PROGRAM P5_00_MAIN
VAR

END_VAR

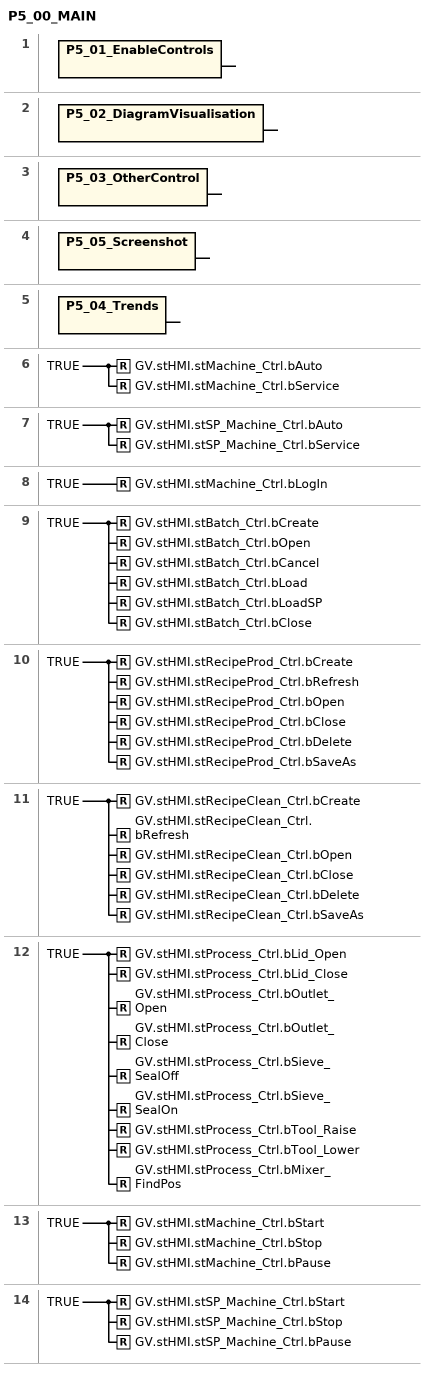
// NETWORK 1
P5_01_EnableControls();

// NETWORK 2
P5_02_DiagramVisualisation();

// NETWORK 3
P5_03_OtherControl();

// NETWORK 4
P5_05_Screenshot();

// NETWORK 5
P5_04_Trends();

// NETWORK 6
GV.stHMI.stMachine_Ctrl.bAuto R= TRUE;
GV.stHMI.stMachine_Ctrl.bService R= TRUE;

// NETWORK 7
GV.stHMI.stSP_Machine_Ctrl.bAuto R= TRUE;
GV.stHMI.stSP_Machine_Ctrl.bService R= TRUE;

// NETWORK 8
GV.stHMI.stMachine_Ctrl.bLogIn R= TRUE;

// NETWORK 9
GV.stHMI.stBatch_Ctrl.bCreate R= TRUE;
GV.stHMI.stBatch_Ctrl.bOpen R= TRUE;
GV.stHMI.stBatch_Ctrl.bCancel R= TRUE;
GV.stHMI.stBatch_Ctrl.bLoad R= TRUE;
GV.stHMI.stBatch_Ctrl.bLoadSP R= TRUE;
GV.stHMI.stBatch_Ctrl.bClose R= TRUE;

// NETWORK 10
GV.stHMI.stRecipeProd_Ctrl.bCreate R= TRUE;
GV.stHMI.stRecipeProd_Ctrl.bRefresh R= TRUE;
GV.stHMI.stRecipeProd_Ctrl.bOpen R= TRUE;
GV.stHMI.stRecipeProd_Ctrl.bClose R= TRUE;
GV.stHMI.stRecipeProd_Ctrl.bDelete R= TRUE;
GV.stHMI.stRecipeProd_Ctrl.bSaveAs R= TRUE;

// NETWORK 11
GV.stHMI.stRecipeClean_Ctrl.bCreate R= TRUE;
GV.stHMI.stRecipeClean_Ctrl.bRefresh R= TRUE;
GV.stHMI.stRecipeClean_Ctrl.bOpen R= TRUE;
GV.stHMI.stRecipeClean_Ctrl.bClose R= TRUE;
GV.stHMI.stRecipeClean_Ctrl.bDelete R= TRUE;
GV.stHMI.stRecipeClean_Ctrl.bSaveAs R= TRUE;

// NETWORK 12
GV.stHMI.stProcess_Ctrl.bLid_Open R= TRUE;
GV.stHMI.stProcess_Ctrl.bLid_Close R= TRUE;
GV.stHMI.stProcess_Ctrl.bOutlet_Open R= TRUE;
GV.stHMI.stProcess_Ctrl.bOutlet_Close R= TRUE;
GV.stHMI.stProcess_Ctrl.bSieve_SealOff R= TRUE;
GV.stHMI.stProcess_Ctrl.bSieve_SealOn R= TRUE;
GV.stHMI.stProcess_Ctrl.bTool_Raise R= TRUE;
GV.stHMI.stProcess_Ctrl.bTool_Lower R= TRUE;
GV.stHMI.stProcess_Ctrl.bMixer_FindPos R= TRUE;

// NETWORK 13
GV.stHMI.stMachine_Ctrl.bStart R= TRUE;
GV.stHMI.stMachine_Ctrl.bStop R= TRUE;
GV.stHMI.stMachine_Ctrl.bPause R= TRUE;

// NETWORK 14
GV.stHMI.stSP_Machine_Ctrl.bStart R= TRUE;
GV.stHMI.stSP_Machine_Ctrl.bStop R= TRUE;
GV.stHMI.stSP_Machine_Ctrl.bPause R= TRUE;

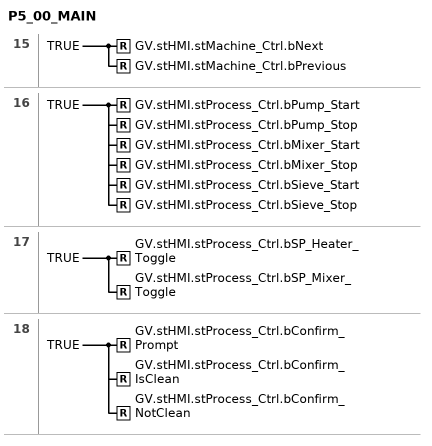
// NETWORK 15
GV.stHMI.stMachine_Ctrl.bNext R= TRUE;
GV.stHMI.stMachine_Ctrl.bPrevious R= TRUE;

// NETWORK 16
GV.stHMI.stProcess_Ctrl.bPump_Start R= TRUE;
GV.stHMI.stProcess_Ctrl.bPump_Stop R= TRUE;
GV.stHMI.stProcess_Ctrl.bMixer_Start R= TRUE;
GV.stHMI.stProcess_Ctrl.bMixer_Stop R= TRUE;
GV.stHMI.stProcess_Ctrl.bSieve_Start R= TRUE;
GV.stHMI.stProcess_Ctrl.bSieve_Stop R= TRUE;

// NETWORK 17
GV.stHMI.stProcess_Ctrl.bSP_Heater_Toggle R= TRUE;
GV.stHMI.stProcess_Ctrl.bSP_Mixer_Toggle R= TRUE;

// NETWORK 18
GV.stHMI.stProcess_Ctrl.bConfirm_Prompt R= TRUE;
GV.stHMI.stProcess_Ctrl.bConfirm_IsClean R= TRUE;
GV.stHMI.stProcess_Ctrl.bConfirm_NotClean R= TRUE;

END_PROGRAM

(* stored: Version 1.1.0.1, ProductVersion 3.1.4024.12
   POU P5_00_MAIN: Id {e5126a8f-d9ae-4302-9246-da3b2a0b21a1}, SpecialFunc None *)
